// TwinCAT 3 PLC project Plc1
// ProgramVersion: 3.1.4024.0
// libraries:
//   Tc2_Standard, * (Beckhoff Automation GmbH)
//   Tc2_System, * (Beckhoff Automation GmbH)
//   Tc3_Module, * (Beckhoff Automation GmbH)
// project tree:
//   / PlcTask.TcTTO
//   POUs/ CalculatePrimeNumbers.TcPOU, MAIN.TcPOU
// real-time tasks:
//   TASK PlcTask: cycle T#10ms, priority 20, ADS port 350

CONFIGURATION Plc1
    RESOURCE PLC ON TwinCAT3
        TASK PlcTask(INTERVAL := T#10ms, PRIORITY := 20);
        PROGRAM MAIN WITH PlcTask : MAIN;
    END_RESOURCE
END_CONFIGURATION

// ---- POUs/MAIN.TcPOU
PROGRAM MAIN
VAR
END_VAR

CalculatePrimeNumbers(10000);

END_PROGRAM

// ---- POUs/CalculatePrimeNumbers.TcPOU
FUNCTION CalculatePrimeNumbers
VAR_INPUT
	n : INT; // Numero di numeri primi da calcolare
END_VAR

VAR
	count : INT := 0; // Contatore per i numeri primi trovati finora
	divisor: INT; // Divisore
	currentNumber : INT := 2; // Numero attuale da verificare
	isPrime : BOOL := TRUE; // Flag che indica se il numero attuale è primo
END_VAR

WHILE count < n DO
	// Verifica se currentNumber è un numero primo
	FOR divisor := 2 TO currentNumber - 1 DO
		IF currentNumber MOD divisor = 0 THEN
			isPrime := FALSE;
			EXIT;
		END_IF
	END_FOR
	
	// Se currentNumber è un numero primo, lo aggiunge all'array
	IF isPrime THEN
		count := count + 1;
	END_IF
	
	// Passa al prossimo numero
	currentNumber := currentNumber + 1;
	isPrime := TRUE; // Reset del flag per il prossimo numero
END_WHILE

END_FUNCTION
